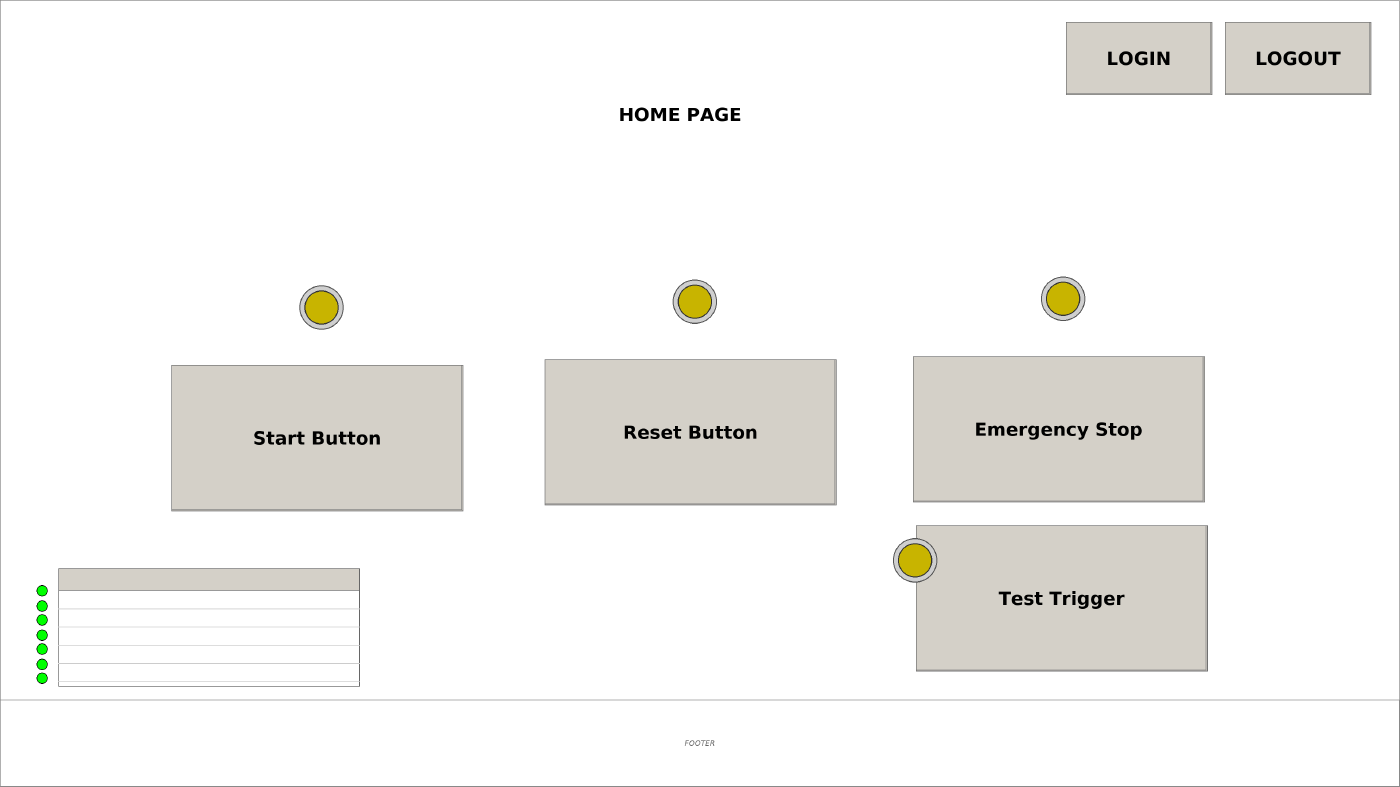
VISUALIZATION PAGE_HOME  // 1920x1080, background image ImagePool.Grey_Gradient
    Button (235,501 400x200), "Start Button"
        OnMouseClick: OpenDialog Dialog=CONFIRMATION, OpenModal=True, OpenCentered=True
    Lamp1 (406,387 70x70), variable: OP_BTN.Start_lamp, style: Lamp-Lamp1-Yellow
    Button (747,493 400x200), "Reset Button"
        tap OP_BTN.Reset_btn
    Lamp1 (918,379 70x70), variable: OP_BTN.Reset_lamp, style: Lamp-Lamp1-Yellow
    Button (1252,489 400x200), "Emergency Stop"
        toggle OP_BTN.Estop_btn
    Lamp1 (1423,375 70x70), variable: OP_BTN.Estop_lamp, style: Lamp-Lamp1-Yellow
    Button (1462,30 200x100), "LOGIN"
        OnMouseClick: VisuUserMgmt Type=Login
    Button (1680,30 200x100), "LOGOUT"
        OnMouseClick: VisuUserMgmt Type=Logout
    Frame (0,960 1920x120)
        shows FOOTER()
    Label (698,99 470x116), "HOME PAGE"
    Table (80,780 413x162), data array: GVL.TableRecord
        p3854506369: GVL.TableRecord[1,INDEX]
        p1892666644: GVL.TableRecord[2,INDEX]
        p338671338: GVL.TableRecord[3,INDEX]
        p2170511999: GVL.TableRecord[4,INDEX]
        p3723444502: GVL.TableRecord[5,INDEX]
        p2232123230: Date
        p511219082: FG-1
        p1755163831: FG-2
        p4092479075: FG-3
        p2237128397: FG-4
    Ellipse (50,803 15x15), invisible if: MAIN.fb_TimeStamp.day[1]
    Ellipse (50,824 15x15), invisible if: MAIN.fb_TimeStamp.day[2]
    Ellipse (50,843 15x15), invisible if: MAIN.fb_TimeStamp.day[3]
    Ellipse (50,864 15x15), invisible if: MAIN.fb_TimeStamp.day[4]
    Ellipse (50,883 15x15), invisible if: MAIN.fb_TimeStamp.day[5]
    Ellipse (50,904 15x15), invisible if: MAIN.fb_TimeStamp.day[6]
    Ellipse (50,923 15x15), invisible if: MAIN.fb_TimeStamp.day[7]
    Button (1256,721 400x200), "Test Trigger"
        toggle OP_BTN.Estop_btn
    Lamp1 (1220,734 70x70), variable: OP_BTN.Estop_lamp, style: Lamp-Lamp1-Yellow
END_VISUALIZATION

(* stored: Version 1.1.0.1, ProductVersion 3.1.4024.12
   Visu PAGE_HOME: Id {d910f869-af87-4472-b9bf-bcfb1b401c7c} *)
